// An incremental hasher that can accept any number of writes.
TYPE blake3_hasher :
STRUCT
  chunk_state					: blake3_chunk_state;
  key_words						: ARRAY[0..7] OF DWORD;
  cv_stack 						: ARRAY[0..8*54] OF DWORD; // Space for 54 subtree chaining values:
  cv_stack_len					: BYTE;      // 2^54 * CHUNK_LEN = 2^64
  flags							: DWORD;
END_STRUCT
END_TYPE

(* stored: Version 1.1.0.1
   DUT blake3_hasher: Id {c277d529-8a84-4560-9ca1-be6281654aca} *)
